{attribute 'qualified_only'}
VAR_GLOBAL CONSTANT
	MAX_NODES : INT := 1000;
END_VAR

(* stored: Version 1.1.0.1, ProductVersion 3.1.4024.12
   GVL GraphFramework: Id {1cdc49ca-6866-01b4-0af3-ddaff08f436e} *)
